// TIA Portal project "红绿灯" (V17)

(* hardware
DEVICE "S7-1200 station_1"  S7-1200 Station
   slot 0: "Rack_0"  S7-1200 Rack  Rack  V1.0
   slot 1: "PLC_1"  CPU 1214C DC/DC/Rly  6ES7 214-1HG40-0XB0  V4.5
*)

// ===== PLC "PLC_1"  CPU 1214C DC/DC/Rly =====

VAR_GLOBAL   // PLC tag table "默认变量表"
   "System_Byte" AT %MB1 : Byte;
   "FirstScan" AT %M1.0 : Bool;
   "DiagStatusUpdate" AT %M1.1 : Bool;
   "AlwaysTRUE" AT %M1.2 : Bool;
   "AlwaysFALSE" AT %M1.3 : Bool;
   "System_Byte(1)" AT %MB1 : Byte;
   "Clock_Byte" AT %MB0 : Byte;
   "Clock_10Hz" AT %M0.0 : Bool;
   "Clock_5Hz" AT %M0.1 : Bool;
   "Clock_2.5Hz" AT %M0.2 : Bool;
   "Clock_2Hz" AT %M0.3 : Bool;
   "Clock_1.25Hz" AT %M0.4 : Bool;
   "Clock_1Hz" AT %M0.5 : Bool;
   "Clock_0.625Hz" AT %M0.6 : Bool;
   "Clock_0.5Hz" AT %M0.7 : Bool;
END_VAR

VAR_GLOBAL   // PLC tag table "输入I"
   "启动按钮" AT %I0.0 : Bool;
END_VAR

VAR_GLOBAL   // PLC tag table "输出Q"
   "红灯" AT %Q0.0 : Bool;
   "绿灯" AT %Q0.1 : Bool;
   "黄灯" AT %Q0.2 : Bool;
END_VAR

DATA_BLOCK "数据块_1"   // DB1
{ S7_Optimized_Access := 'TRUE' }
VERSION : 0.1
   VAR
      进入循环 : Bool;
      当前时间_0 : Time;
      红灯程序 : Bool;
      绿灯程序 : Bool;
      黄灯程序 : Bool;
      当前时间_1 : Time;
      当前时间_2 : Time;
      红灯结束 : Bool;
      绿灯结束 : Bool;
      黄灯结束 : Bool;
      三次结束 : Bool;
      nexttime : Bool;
      结束程序 : Bool;
   END_VAR
BEGIN
END_DATA_BLOCK

// folder: System blocks/Program resources

DATA_BLOCK "IEC_Timer_0_DB"   // DB2
{ S7_Optimized_Access := 'TRUE' }
AUTHOR : Simatic
FAMILY : IEC
NAME : IEC_TMR
VERSION : 1.0
// stored: InstanceOfName IEC_TIMER
"IEC_TIMER"
BEGIN
END_DATA_BLOCK

DATA_BLOCK "IEC_Timer_0_DB_1"   // DB3
{ S7_Optimized_Access := 'TRUE' }
AUTHOR : Simatic
FAMILY : IEC
NAME : IEC_TMR
VERSION : 1.0
// stored: InstanceOfName IEC_TIMER
"IEC_TIMER"
BEGIN
END_DATA_BLOCK

DATA_BLOCK "IEC_Timer_0_DB_2"   // DB4
{ S7_Optimized_Access := 'TRUE' }
AUTHOR : Simatic
FAMILY : IEC
NAME : IEC_TMR
VERSION : 1.0
// stored: InstanceOfName IEC_TIMER
"IEC_TIMER"
BEGIN
END_DATA_BLOCK

DATA_BLOCK "IEC_Counter_0_DB_1"   // DB6
{ S7_Optimized_Access := 'TRUE' }
AUTHOR : Simatic
FAMILY : IEC
NAME : CNTR
VERSION : 1.0
// stored: InstanceOfName IEC_COUNTER
"IEC_COUNTER"
BEGIN
END_DATA_BLOCK

// folder: (top level)

ORGANIZATION_BLOCK "Main"   // OB1, LAD, ProgramCycle
TITLE = "Main Program Sweep (Cycle)"
{ S7_Optimized_Access := 'TRUE' }
VERSION : 0.1
   VAR_INPUT
      Initial_Call : Bool;   // Initial call of this OB
      Remanence : Bool;   // =True, if remanent data are available
   END_VAR
BEGIN

REGION Network 1: 启动程序
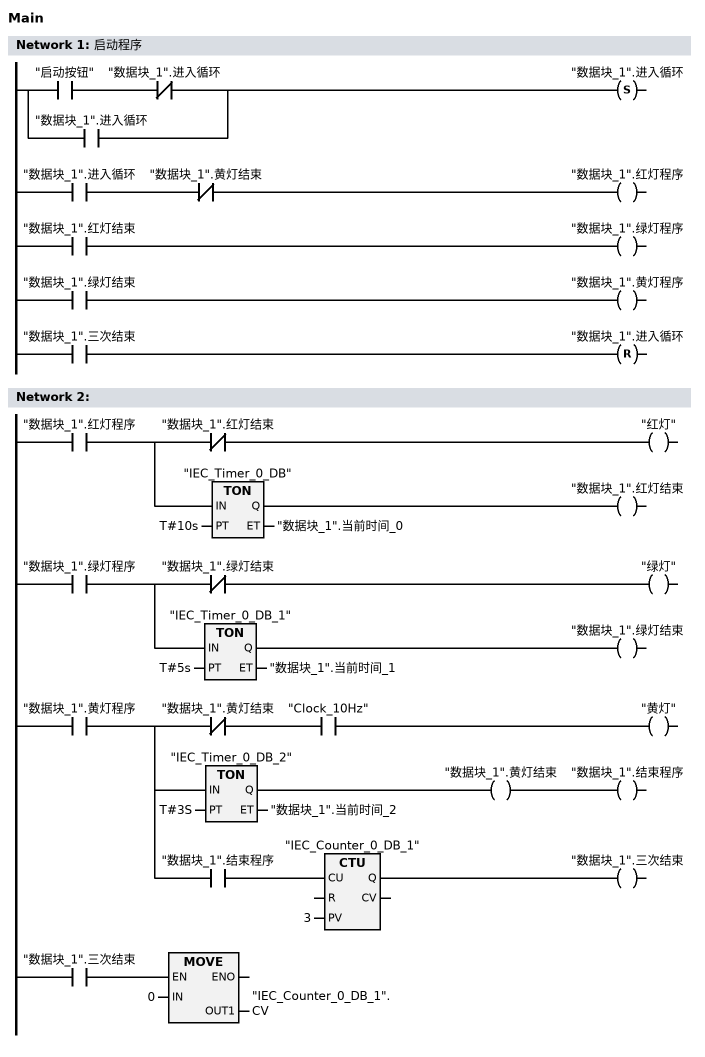
   RUNG wire#powerrail
      Contact( "启动按钮" )
      I_Contact( "数据块_1".进入循环 )
      wire#w1
      S_Coil( "数据块_1".进入循环 )
   END_RUNG
   RUNG wire#powerrail
      Contact( "数据块_1".进入循环 )
   END_RUNG wire#w1
   RUNG wire#powerrail
      Contact( "数据块_1".进入循环 )
      I_Contact( "数据块_1".黄灯结束 )
      Coil( "数据块_1".红灯程序 )
   END_RUNG
   RUNG wire#powerrail
      Contact( "数据块_1".红灯结束 )
      Coil( "数据块_1".绿灯程序 )
   END_RUNG
   RUNG wire#powerrail
      Contact( "数据块_1".绿灯结束 )
      Coil( "数据块_1".黄灯程序 )
   END_RUNG
   RUNG wire#powerrail
      Contact( "数据块_1".三次结束 )
      R_Coil( "数据块_1".进入循环 )
   END_RUNG
   // the same network as SCL:
   IF ("启动按钮" AND NOT "数据块_1".进入循环) OR "数据块_1".进入循环 THEN "数据块_1".进入循环 := TRUE; END_IF;
   "数据块_1".红灯程序 := "数据块_1".进入循环 AND NOT "数据块_1".黄灯结束;
   "数据块_1".绿灯程序 := "数据块_1".红灯结束;
   "数据块_1".黄灯程序 := "数据块_1".绿灯结束;
   IF "数据块_1".三次结束 THEN "数据块_1".进入循环 := FALSE; END_IF;
END_REGION

REGION Network 2
   "红灯" := "数据块_1".红灯程序 AND NOT "数据块_1".红灯结束;
   "IEC_Timer_0_DB".TON(IN := "数据块_1".红灯程序, PT := T#10s, ET => "数据块_1".当前时间_0);
   "数据块_1".红灯结束 := "IEC_Timer_0_DB".Q;
   "绿灯" := "数据块_1".绿灯程序 AND NOT "数据块_1".绿灯结束;
   "IEC_Timer_0_DB_1".TON(IN := "数据块_1".绿灯程序, PT := T#5s, ET => "数据块_1".当前时间_1);
   "数据块_1".绿灯结束 := "IEC_Timer_0_DB_1".Q;
   "黄灯" := "数据块_1".黄灯程序 AND NOT "数据块_1".黄灯结束 AND "Clock_10Hz";
   "IEC_Timer_0_DB_2".TON(IN := "数据块_1".黄灯程序, PT := T#3S, ET => "数据块_1".当前时间_2);
   "数据块_1".黄灯结束 := "IEC_Timer_0_DB_2".Q;
   "数据块_1".结束程序 := "IEC_Timer_0_DB_2".Q;
   "IEC_Counter_0_DB_1".CTU(CU := "数据块_1".黄灯程序 AND "数据块_1".结束程序, PV := 3);
   "数据块_1".三次结束 := "IEC_Counter_0_DB_1".Q;
   IF "数据块_1".三次结束 THEN "IEC_Counter_0_DB_1".CV := 0; END_IF;
END_REGION
END_ORGANIZATION_BLOCK